// TwinCAT 3 PLC project PLCTesting
// ProgramVersion: 3.1.4024.0
// libraries:
//   Tc2_Standard, * (Beckhoff Automation GmbH)
//   Tc2_System, * (Beckhoff Automation GmbH)
//   Tc3_Module, * (Beckhoff Automation GmbH)
// project tree:
//   DUTs/ E_MachineConditions.TcDUT, SensorBrands.TcDUT, ST_MachineOperatingParameters.TcDUT, ST_MotorParameters.TcDUT, ST_Timer.TcDUT
//   / GlobalTextList.TcGTLO, PlcTask.TcTTO, PlcTaskRef.TcTTO, Visualization Manager.TcVMO (not stored)
//   GVLs/ GVL_Task1.TcGVL, GVL_Task2.TcGVL, GVL_Task3.TcGVL
//   POUs/ F_IncreaseTemperature.TcPOU, F_DecreaseTemperature.TcPOU, F_UpdateParameter.TcPOU, F_UpdateParameterRef.TcPOU, MAIN.TcPOU, PLC_Task1.TcPOU, PLC_Task2.TcPOU, PLC_Task3.TcPOU, PLC_TaskCase.TcPOU, RadToDeg.TcPOU
//   VISUs/ Visualization.TcVIS

CONFIGURATION PLCTesting
    RESOURCE PLC ON TwinCAT3
        TASK PlcTask(INTERVAL := T#10ms, PRIORITY := 20);
        TASK PlcTaskRef(INTERVAL := T#10ms, PRIORITY := 1);
        PROGRAM MAIN WITH PlcTask : MAIN;
        PROGRAM PLC_TaskCase WITH PlcTaskRef : PLC_TaskCase;
    END_RESOURCE
END_CONFIGURATION

// ---- DUTs/E_MachineConditions.TcDUT
{attribute 'qualified_only'}
{attribute 'strict'}
TYPE E_MachineConditions :
(
	unIsReadyToStart := 0,
	unIsHeating := 1,
	unIsSmelting := 2,
	unIsCooling := 3
)UINT;
END_TYPE

// ---- DUTs/SensorBrands.TcDUT
{attribute 'qualified_only'}
{attribute 'strict'}
TYPE SensorBrands :
(
 	Sick := 0,
	Pilz := 1,
	Parker := 2,
	Bosch := 3	
);
END_TYPE

// ---- DUTs/ST_MachineOperatingParameters.TcDUT
TYPE ST_MachineOperatingParameters :
STRUCT
	unCurrentState : UINT;
	bStartButtonPressed : BOOL;
	fTemperature : REAL;
	
	bIsHeating : BOOL;
	bIsSmelting : BOOL;
	bIsCooling : BOOL;
	
	tTimeToHeat : TIME := T#5S;
	tTimeToSmelt : TIME := T#5S;
	tTimeToCool : TIME := T#10S;
	
	fHeatingConstant : REAL := 0.1; // Degree / Cycle time (1ms)
	fCoolingConstant : REAL := 0.05; // Degree / Cycle time (1ms)
	
END_STRUCT
END_TYPE

// ---- DUTs/ST_MotorParameters.TcDUT
TYPE ST_MotorParameters :
	
STRUCT
	
fMinSpeed : REAL;
fMaxSpeed : REAL;

END_STRUCT

END_TYPE

// ---- DUTs/ST_Timer.TcDUT
TYPE ST_Timer:
	
STRUCT
	bStart : BOOL;
	tTime : TIME := T#10S;
	tElapsedTime : TIME;
	bQ : BOOL;
END_STRUCT

END_TYPE

// ---- GVLs/GVL_Task1.TcGVL
{attribute 'qualified_only'}
VAR_GLOBAL
	dtThisIsADTVariable : DATE_AND_TIME := DT#2024-02-26-12:07:05;
	nThisIsAnInteger : INT := 30;
	dThisIsADateArray : ARRAY[0..3] OF DATE := [D#2024-02-26, D#2024-02-27, D#2024-02-28, D#2024-02-29];
	
	bStart : BOOL;
	tTime : TIME := T#10S;
	tElapsedTime : TIME;
	bQ : BOOL;
	
END_VAR

// ---- GVLs/GVL_Task2.TcGVL
{attribute 'qualified_only'}
VAR_GLOBAL
	stTimer : ST_Timer := (tTime := T#5S);
	fMotor1Rad : REAL;
	fMotor1Deg : REAL;
END_VAR

// ---- GVLs/GVL_Task3.TcGVL
{attribute 'qualified_only'}
VAR_GLOBAL
	stMotor1 : ST_MotorParameters;
	stMotor2 : ST_MotorParameters;
END_VAR

// ---- POUs/MAIN.TcPOU
PROGRAM MAIN
VAR
END_VAR

END_PROGRAM

// ---- POUs/PLC_TaskCase.TcPOU
PROGRAM PLC_TaskCase
VAR
	stMachine1 : ST_MachineOperatingParameters;
	tCycleTime : REAL := 10.0; // ms
	
	fbRTrig : R_TRIG;
	bStart : BOOL;
	
	tonTimerHeating : TON;
	tonTimerSmelting : TON;
	tonTimerCooling : TON;
	
	
	
END_VAR

CASE stMachine1.unCurrentState OF
	
	E_MachineConditions.unIsReadyToStart:		
		fbRTrig(CLK := stMachine1.bStartButtonPressed, Q => bStart);
		
		IF bStart THEN
			stMachine1.unCurrentState := E_MachineConditions.unIsHeating;
		END_IF
		
		
	E_MachineConditions.unIsHeating: //////////////////////////
		stMachine1.bIsHeating := TRUE;
		
		tonTimerHeating(
		IN := stMachine1.bIsHeating, 
		PT := stMachine1.tTimeToHeat);
		
		IF tonTimerHeating.ET < stMachine1.tTimeToHeat THEN
			F_IncreaseTemperature(stMachine := stMachine1, tCycleTime := tCycleTime);
		END_IF
		
		IF tonTimerHeating.Q = TRUE THEN
			tonTimerHeating(IN := FALSE); // Resets the TON timer for heating, since this is the next cycle
			stMachine1.bIsHeating := FALSE; // Is not heating anymore
			stMachine1.unCurrentState := E_MachineConditions.unIsSmelting;
		END_IF
		
		
	
	E_MachineConditions.unIsSmelting: /////////////////
		
		stMachine1.bIsSmelting := TRUE;
		
		tonTimerSmelting(
		IN := stMachine1.bIsSmelting, 
		PT := stMachine1.tTimeToSmelt);
		
		IF tonTimerSmelting.ET < stMachine1.tTimeToSmelt THEN
			stMachine1.fTemperature := stMachine1.fTemperature;
		END_IF
		
		IF tonTimerSmelting.Q = TRUE THEN
			tonTimerSmelting(IN := FALSE); // Resets the TON timer for smelting, since this is the next cycle
			stMachine1.bIsSmelting := FALSE; // Is not smelting anymore
			stMachine1.unCurrentState := E_MachineConditions.unIsCooling;
		END_IF
	
		
		E_MachineConditions.unIsCooling: //////////////
		
		stMachine1.bIsCooling := TRUE;
		
		tonTimerCooling(
		IN := stMachine1.bIsCooling, 
		PT := stMachine1.tTimeToCool);
		
		IF tonTimerCooling.ET < stMachine1.tTimeToCool THEN
			F_DecreaseTemperature(stMachine := stMachine1, tCycleTime := tCycleTime);
		END_IF
		
		IF tonTimerCooling.Q = TRUE THEN
			tonTimerCooling(IN := FALSE); // Resets the TON timer for cooling, since it ends here next cycle
			stMachine1.bIsCooling := FALSE; // Is not cooling anymore
			stMachine1.unCurrentState := E_MachineConditions.unIsReadyToStart;
			bStart := FALSE;
		END_IF
			
END_CASE

END_PROGRAM

// ---- POUs/F_IncreaseTemperature.TcPOU
FUNCTION F_IncreaseTemperature

VAR_INPUT
	stMachine : REFERENCE TO ST_MachineOperatingParameters;
	tCycleTime : REAL;
END_VAR

VAR
END_VAR

stMachine.fTemperature := stMachine.fTemperature + (stMachine.fHeatingConstant * tCycleTime);

END_FUNCTION

// ---- POUs/F_DecreaseTemperature.TcPOU
FUNCTION F_DecreaseTemperature

VAR_INPUT
	stMachine : REFERENCE TO ST_MachineOperatingParameters;
	tCycleTime : REAL;
END_VAR

VAR
END_VAR

stMachine.fTemperature := stMachine.fTemperature - (stMachine.fCoolingConstant * tCycleTime);

END_FUNCTION

// ---- POUs/F_UpdateParameter.TcPOU
FUNCTION F_UpdateParameter
VAR_INPUT
	bUpdateValue : BOOL;
	fNewValue : REAL;
	stMotorParameters : ST_MotorParameters;
END_VAR

VAR_OUTPUT
	stMotorParametersUpdated : ST_MotorParameters;
END_VAR

IF bUpdateValue THEN
	stMotorParametersUpdated.fMaxSpeed := fNewValue;
ELSE
	stMotorParametersUpdated.fMaxSpeed := stMotorParameters.fMaxSpeed;	
END_IF

END_FUNCTION

// ---- POUs/F_UpdateParameterRef.TcPOU
FUNCTION F_UpdateParameterRef
VAR_INPUT
	bUpdateValue : BOOL;
	fNewValue : REAL;
	stMotorParameters : REFERENCE TO ST_MotorParameters;
END_VAR

VAR
END_VAR

IF bUpdateValue THEN
	stMotorParameters.fMaxSpeed := fNewValue;
ELSE
	stMotorParameters.fMaxSpeed := stMotorParameters.fMaxSpeed;	
END_IF

END_FUNCTION

// ---- POUs/PLC_Task1.TcPOU
PROGRAM PLC_Task1
VAR
	dtPointer : POINTER TO DATE_AND_TIME;
	nPointer : POINTER TO INT;
	
	dtReference : REFERENCE TO DATE_AND_TIME;
	nReference : REFERENCE TO INT;
	
	sensor1 : INT;
	
	tonTimer : TON;
END_VAR

dtPointer := ADR(GVL_Task1.dtThisIsADTVariable);
dtPointer^ := DT#2025-12-12-12:30:30;

nPointer := ADR(GVL_Task1.nThisIsAnInteger);
nPointer^ := 40;

dtReference REF=GVL_Task1.dtThisIsADTVariable;
nReference REF=GVL_Task1.nThisIsAnInteger;

dtReference := DT#2025-12-12-12:30:31;
nReference := 70;

GVL_Task1.dThisIsADateArray[3] := D#2024-02-04;

sensor1 := SensorBrands.Parker;

tonTimer(IN := GVL_Task1.bStart, PT := GVL_Task1.tTime, Q => GVL_Task1.bQ, ET => GVL_Task1.tElapsedTime);

END_PROGRAM

// ---- POUs/PLC_Task2.TcPOU
PROGRAM PLC_Task2
VAR
	tofTimer : TOF;
END_VAR

tofTimer(IN := GVL_Task2.stTimer.bStart, PT := GVL_Task2.stTimer.tTime, Q => GVL_Task2.stTimer.bQ, ET => GVL_Task2.stTimer.tElapsedTime);

GVL_Task2.fMotor1Rad := 2.0;
RadToDeg(GVL_Task2.fMotor1Rad, fAngleDeg => GVL_Task2.fMotor1Deg);

END_PROGRAM

// ---- POUs/RadToDeg.TcPOU
FUNCTION RadToDeg : REAL

VAR_INPUT
	fAngle : REAL;
END_VAR

VAR
	fRadToDegConstant : REAL := 57.295;
END_VAR

VAR_OUTPUT
	fAngleDeg : REAL;
END_VAR


fAngleDeg := fAngle * fRadToDegConstant;

END_FUNCTION

// ---- POUs/PLC_Task3.TcPOU
PROGRAM PLC_Task3
VAR
	fbRTrig : R_TRIG;
	bBoolean : BOOL;
	bQ : BOOL;
	fNewSpeed : REAL := 40.0;
END_VAR

fbRTrig(CLK := bBoolean, Q => bQ);

GVL_Task3.stMotor1 := F_UpdateParameter
(
bUpdateValue := bQ, 
fNewValue := fNewSpeed,
stMotorParameters := GVL_Task3.stMotor1
);

F_UpdateParameterRef
(
bUpdateValue := bQ, 
fNewValue := fNewSpeed, 
stMotorParameters := GVL_Task3.stMotor2
);

END_PROGRAM

// ---- GlobalTextList.TcGTLO
TEXTLIST GlobalTextList
  277 = 'Controls'
END_TEXTLIST

// ---- VISUs/Visualization.TcVIS
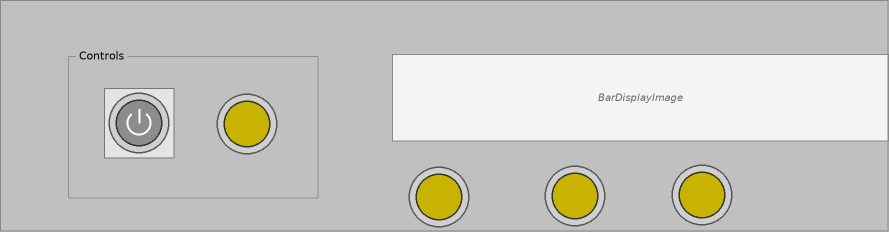
VISUALIZATION Visualization  // 889x232
    BarDisplayImage (392,54 497x87), value: PLC_TaskCase.stMachine1.fTemperature, style: BarDisplayImage-Gray, scale format: %.1f, scale 0..500
    GroupBox (68,48 250x150), "Controls"
        Lamp1 (144,41 70x70), variable: PLC_TaskCase.bStart, style: Lamp-Lamp1-Yellow
        PowerSwitch (36,40 70x70), variable: PLC_TaskCase.stMachine1.bStartButtonPressed, behaviour: TOGGLE, style: Switch-PowerSwitch-Gray
    Lamp1 (667,160 70x70), variable: PLC_TaskCase.stMachine1.bIsCooling, style: Lamp-Lamp1-Yellow
    Lamp1 (540,161 70x70), variable: PLC_TaskCase.stMachine1.bIsSmelting, style: Lamp-Lamp1-Yellow
    Lamp1 (404,162 70x70), variable: PLC_TaskCase.stMachine1.bIsHeating, style: Lamp-Lamp1-Yellow
END_VISUALIZATION
